INTERFACE I_MaintenanceMode EXTENDS I_PackMLMode

END_INTERFACE

(* stored: Version 1.1.0.1, ProductVersion 3.1.4024.12
   Itf I_MaintenanceMode: Id {3db8b67a-88f5-4699-963d-be2fe99617ef} *)
